FUNCTION_BLOCK CylControl (* Basic Function Block Type *)
  (* Standard: 61499-2 *)
  (* Version 0.0, 11/30/2015, paarnio, nxtControl GmbH, Template *)
  PACKAGE Main;
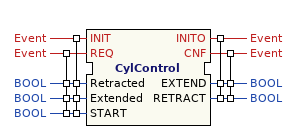
  EVENT_INPUT
    INIT WITH Retracted, Extended, START; (* Initialization Request *)
    REQ WITH Retracted, Extended, START; (* Normal Execution Request *)
  END_EVENT
  EVENT_OUTPUT
    INITO WITH EXTEND, RETRACT; (* Initialization Confirm *)
    CNF WITH EXTEND, RETRACT; (* Execution Confirmation *)
  END_EVENT
  VAR_INPUT
    Retracted : BOOL;
    Extended : BOOL;
    START : BOOL;
  END_VAR
  VAR_OUTPUT
    EXTEND : BOOL;
    RETRACT : BOOL;
  END_VAR
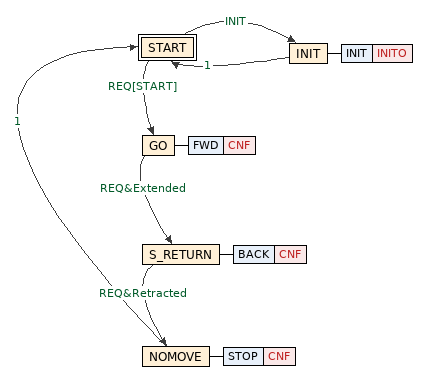
  EC_STATES
    START; (* Initial State *)
    INIT : INIT -> INITO; (* Initialization *)
    GO : FWD -> CNF;
    S_RETURN : BACK -> CNF;
    NOMOVE : STOP -> CNF;
  END_STATES
  EC_TRANSITIONS
    START TO INIT := INIT;
    INIT TO START := 1;
    START TO GO := REQ[START];
    GO TO S_RETURN := REQ&Extended;
    S_RETURN TO NOMOVE := REQ&Retracted;
    NOMOVE TO START := 1;
  END_TRANSITIONS
  ALGORITHM INIT IN ST: (* Initialization algorithm *)
EXTEND:=FALSE;
RETRACT:=FALSE;
  END_ALGORITHM
  ALGORITHM REQ IN ST: (* Normally executed algorithm *)
;
  END_ALGORITHM
  ALGORITHM FWD IN ST:
EXTEND:=TRUE;
RETRACT:=FALSE;
  END_ALGORITHM
  ALGORITHM BACK IN ST:
EXTEND:=FALSE;
RETRACT:=TRUE;
  END_ALGORITHM
  ALGORITHM STOP IN ST:
EXTEND:=FALSE;
RETRACT:=FALSE;
  END_ALGORITHM
END_FUNCTION_BLOCK
